INTERFACE IRfidTasks

METHOD ReadUid : BOOL
VAR_INPUT
END_VAR
END_METHOD

END_INTERFACE

(* stored: Version 1.1.0.1, ProductVersion 3.1.4024.12
   Itf IRfidTasks: Id {26a272db-a857-0f88-2252-988e3d5e5b9a}
   Method ReadUid: Id {feea7b61-9dc9-0e14-11a3-c805fd5a4db1} *)
